FUNCTION_BLOCK FB_Cylinder_Test EXTENDS TcUnit.FB_TestSuite
VAR
	fbCylinder : FB_Cylinder;
	nExpected : BYTE;
	nResult : BYTE;
	bExpected : BOOL;
	bResult : BOOL;
END_VAR

TEST('bRetract FALSE');
fbCylinder.bRetract := FALSE;
fbCylinder();
bExpected := FALSE;
nResult := fbCylinder.GetControl();
bResult := nResult.0;

AssertEquals(Expected := bExpected,
             Actual := bResult,
             Message := 'Control value is not correct');	
TEST_FINISHED();

TEST('bRetract TRUE');
fbCylinder.bRetract := TRUE;
fbCylinder();
bExpected := TRUE;
nResult := fbCylinder.GetControl();
bResult := nResult.0;

AssertEquals(Expected := bExpected,
             Actual := bResult,
             Message := 'Control value is not correct');	
TEST_FINISHED();

TEST('bExtend FALSE');
fbCylinder.bExtend := FALSE;
fbCylinder();
bExpected := FALSE;
nResult := fbCylinder.GetControl();
bResult := nResult.1;

AssertEquals(Expected := bExpected,
             Actual := bResult,
             Message := 'Control value is not correct');	
TEST_FINISHED();

TEST('bExtend TRUE');
fbCylinder.bExtend := TRUE;
fbCylinder();
bExpected := TRUE;
nResult := fbCylinder.GetControl();
bResult := nResult.1;

AssertEquals(Expected := bExpected,
             Actual := bResult,
             Message := 'Control value is not correct');	
TEST_FINISHED();

TEST('bRetracted FALSE');
fbCylinder.SetStatus(0);
fbCylinder();
bExpected := FALSE;
bResult := fbCylinder.bRetracted;

AssertEquals(Expected := bExpected,
             Actual := bResult,
             Message := 'Control value is not correct');	
TEST_FINISHED();

TEST('bRetracted TRUE');
fbCylinder.SetStatus(1);
fbCylinder();
bExpected := TRUE;
bResult := fbCylinder.bRetracted;

AssertEquals(Expected := bExpected,
             Actual := bResult,
             Message := 'Control value is not correct');	
TEST_FINISHED();

TEST('bExtended FALSE');
fbCylinder.SetStatus(0);
fbCylinder();
bExpected := FALSE;
bResult := fbCylinder.bExtended;

AssertEquals(Expected := bExpected,
             Actual := bResult,
             Message := 'Control value is not correct');	
TEST_FINISHED();

TEST('bExtended TRUE');
fbCylinder.SetStatus(2);
fbCylinder();
bExpected := TRUE;
bResult := fbCylinder.bExtended;

AssertEquals(Expected := bExpected,
             Actual := bResult,
             Message := 'Control value is not correct');	
TEST_FINISHED();

END_FUNCTION_BLOCK

(* stored: Version 1.1.0.1, ProductVersion 3.1.4024.12
   POU FB_Cylinder_Test: Id {4aa5bec3-e8a9-0d97-0520-d08e52c6fe69}, SpecialFunc None *)
